// TIA Portal V18 export
ORGANIZATION_BLOCK "21-SafetyShoe"   // OB134, LAD, ProgramCycle
TITLE = "Main Program Sweep (Cycle)"
{ S7_Optimized_Access := 'TRUE' }
VERSION : 0.1
// stored: AutoNumber true, IsIECCheckEnabled false, SetENOAutomatically false
   VAR_INPUT
      Initial_Call : Bool;   // Initial call of this OB
      Remanence : Bool;   // =True, if remanent data are available
   END_VAR
   VAR_TEMP   // added for the SCL form of the ladder/FBD networks
      _w1 : Bool;
   END_VAR
BEGIN

REGION Network 1: SafetyShoe
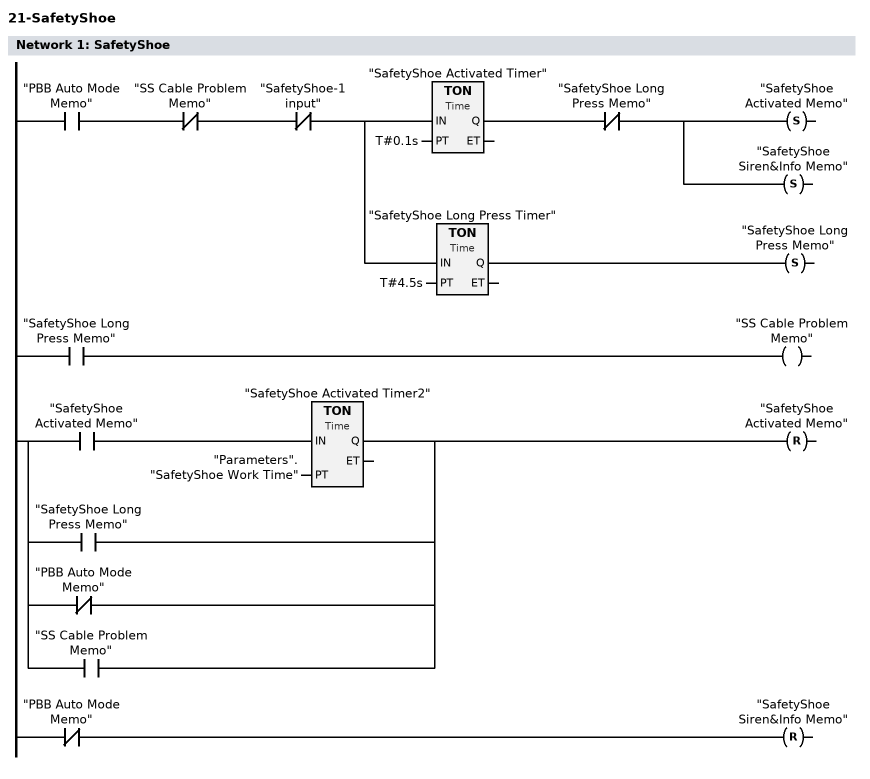
   RUNG wire#powerrail
      Contact( "PBB Auto Mode Memo" )
      I_Contact( "SS Cable Problem Memo" )
      I_Contact( "SafetyShoe-1 input" )
      wire#w1
      { S7_Templates := "time_type := Time" } "SafetyShoe Activated Timer".TON(pt := T#0.1s, et =>)
      I_Contact( "SafetyShoe Long Press Memo" )
      wire#w2
      S_Coil( "SafetyShoe Activated Memo" )
   END_RUNG
   RUNG wire#w2
      S_Coil( "SafetyShoe Siren&Info Memo" )
   END_RUNG
   RUNG wire#w1
      { S7_Templates := "time_type := Time" } "SafetyShoe Long Press Timer".TON(pt := T#4.5s, et =>)
      S_Coil( "SafetyShoe Long Press Memo" )
   END_RUNG
   RUNG wire#powerrail
      Contact( "SafetyShoe Long Press Memo" )
      Coil( "SS Cable Problem Memo" )
   END_RUNG
   RUNG wire#powerrail
      Contact( "SafetyShoe Activated Memo" )
      { S7_Templates := "time_type := Time" } "SafetyShoe Activated Timer2".TON(pt := "Parameters"."SafetyShoe Work Time", et =>)
      wire#w3
      R_Coil( "SafetyShoe Activated Memo" )
   END_RUNG
   RUNG wire#powerrail
      Contact( "SafetyShoe Long Press Memo" )
   END_RUNG wire#w3
   RUNG wire#powerrail
      I_Contact( "PBB Auto Mode Memo" )
   END_RUNG wire#w3
   RUNG wire#powerrail
      Contact( "SS Cable Problem Memo" )
   END_RUNG wire#w3
   RUNG wire#powerrail
      I_Contact( "PBB Auto Mode Memo" )
      R_Coil( "SafetyShoe Siren&Info Memo" )
   END_RUNG
   // the same network as SCL:
   #_w1 := "PBB Auto Mode Memo" AND NOT "SS Cable Problem Memo" AND NOT "SafetyShoe-1 input";
   "SafetyShoe Activated Timer".TON(IN := #_w1, PT := T#0.1s);
   IF "SafetyShoe Activated Timer".Q AND NOT "SafetyShoe Long Press Memo" THEN
       "SafetyShoe Activated Memo" := TRUE;
       "SafetyShoe Siren&Info Memo" := TRUE;
   END_IF;
   "SafetyShoe Long Press Timer".TON(IN := #_w1, PT := T#4.5s);
   IF "SafetyShoe Long Press Timer".Q THEN "SafetyShoe Long Press Memo" := TRUE; END_IF;
   "SS Cable Problem Memo" := "SafetyShoe Long Press Memo";
   "SafetyShoe Activated Timer2".TON(IN := "SafetyShoe Activated Memo",
                           PT := "Parameters"."SafetyShoe Work Time");
   IF "SafetyShoe Activated Timer2".Q OR "SafetyShoe Long Press Memo" OR NOT "PBB Auto Mode Memo" OR "SS Cable Problem Memo" THEN
       "SafetyShoe Activated Memo" := FALSE;
   END_IF;
   IF NOT "PBB Auto Mode Memo" THEN "SafetyShoe Siren&Info Memo" := FALSE; END_IF;
END_REGION
END_ORGANIZATION_BLOCK
